// TIA Portal V18 export
// export: Created 2026-06-12T02:00:00Z, ExportSetting WithDefaults, DisplayName Totally Integrated Automation Portal, DisplayVersion V18, DisplayName TIA Portal Openness, DisplayVersion V18
TagTable "AI_B5_Tags"
  AI_B5_CA_Fan_Motor_DE_Temp : Real  (PLC tag AI_B5_CA_Fan_Motor_DE_Temp, HMI_Connection_1, 1 s)   // TEMP 50-80 °C
  AI_B5_CA_Fan_Motor_NDE_Temp : Real  (PLC tag AI_B5_CA_Fan_Motor_NDE_Temp, HMI_Connection_1, 1 s)   // TEMP 50-80 °C
  AI_B5_CA_Fan_DE_Temp : Real  (PLC tag AI_B5_CA_Fan_DE_Temp, HMI_Connection_1, 1 s)   // TEMP 50-80 °C
  AI_B5_CA_Fan_NDE_Temp : Real  (PLC tag AI_B5_CA_Fan_NDE_Temp, HMI_Connection_1, 1 s)   // TEMP 50-80 °C
  AI_B5_CA_Fan_DE_Vib : Real  (PLC tag AI_B5_CA_Fan_DE_Vib, HMI_Connection_1, 1 s)   // COUNT 0-10 mm/s
  AI_B5_CA_Fan_NDE_Vib : Real  (PLC tag AI_B5_CA_Fan_NDE_Vib, HMI_Connection_1, 1 s)   // COUNT 0-10 mm/s
  AI_B5_SP_700FN03 : Real  (PLC tag AI_B5_SP_700FN03, HMI_Connection_1, 1 s)   // FLOW 100-200 L/h
  AI_B5_SP_700HES01 : Real  (PLC tag AI_B5_SP_700HES01, HMI_Connection_1, 1 s)   // FLOW 100-200 L/h
  AI_B5_SP_700DA4 : Real  (PLC tag AI_B5_SP_700DA4, HMI_Connection_1, 1 s)   // FREQ 20-30 Hz
  AI_B5_SP_700DA6 : Real  (PLC tag AI_B5_SP_700DA6, HMI_Connection_1, 1 s)   // FREQ 20-30 Hz
  AI_B5_SP_700DA7 : Real  (PLC tag AI_B5_SP_700DA7, HMI_Connection_1, 1 s)   // FREQ 20-30 Hz
  AI_B5_SP_700FN2_DA1 : Real  (PLC tag AI_B5_SP_700FN2_DA1, HMI_Connection_1, 1 s)   // FREQ 20-30 Hz
  AI_B5_Sep_Motor_Top_Temp : Real  (PLC tag AI_B5_Sep_Motor_Top_Temp, HMI_Connection_1, 1 s)   // TEMP 50-80 °C
  AI_B5_Sep_Bottom_Bear_Temp : Real  (PLC tag AI_B5_Sep_Bottom_Bear_Temp, HMI_Connection_1, 1 s)   // TEMP 50-80 °C
  AI_B5_Trend_Val_1 : Real  (PLC tag AI_B5_Trend_Val_1, HMI_Connection_1, 1 s)   // PERCENT 0-100 %
  AI_B5_Trend_Val_2 : Real  (PLC tag AI_B5_Trend_Val_2, HMI_Connection_1, 1 s)   // PERCENT 0-100 %
  AI_B5_Trend_Val_3 : Real  (PLC tag AI_B5_Trend_Val_3, HMI_Connection_1, 1 s)   // PERCENT 0-100 %
  AI_B5_700FN03_RPM : Real  (PLC tag AI_B5_700FN03_RPM, HMI_Connection_1, 1 s)   // RPM 800-1200 RPM
  AI_B5_700HES01_Flow : Real  (PLC tag AI_B5_700HES01_Flow, HMI_Connection_1, 1 s)   // FLOW 100-200 L/h
  AI_B5_700FN10_Speed : Real  (PLC tag AI_B5_700FN10_Speed, HMI_Connection_1, 1 s)   // FREQ 20-30 Hz
  AI_B5_700CM01_Current : Real  (PLC tag AI_B5_700CM01_Current, HMI_Connection_1, 1 s)   // CURRENT 50-200 A
  AI_B5_Lub_Stop_Time : Real  (PLC tag AI_B5_Lub_Stop_Time, HMI_Connection_1, 1 s)   // COUNT 0-300 Sec
  AI_B5_Main_Drive_ReHealth : Real  (PLC tag AI_B5_Main_Drive_ReHealth, HMI_Connection_1, 1 s)   // COUNT 0-300 Sec
  AI_B5_CM_LRS_IN : Real  (PLC tag AI_B5_CM_LRS_IN, HMI_Connection_1, 1 s)   // TEMP 50-80 °C
  AI_B5_CM_LRS_OUT : Real  (PLC tag AI_B5_CM_LRS_OUT, HMI_Connection_1, 1 s)   // TEMP 50-80 °C
  AI_B5_CM_Mill_Oil_Temp : Real  (PLC tag AI_B5_CM_Mill_Oil_Temp, HMI_Connection_1, 1 s)   // TEMP 50-80 °C
  AI_B5_CM_OilTrun_BER_Temp : Real  (PLC tag AI_B5_CM_OilTrun_BER_Temp, HMI_Connection_1, 1 s)   // TEMP 50-80 °C
  AI_B5_CM_OilTrun_BER2_Temp : Real  (PLC tag AI_B5_CM_OilTrun_BER2_Temp, HMI_Connection_1, 1 s)   // TEMP 50-80 °C
  AI_B5_CM_OilPinion_BER_Temp : Real  (PLC tag AI_B5_CM_OilPinion_BER_Temp, HMI_Connection_1, 1 s)   // TEMP 50-80 °C
  AI_B5_CM_GB_IL_Shaft_BER : Real  (PLC tag AI_B5_CM_GB_IL_Shaft_BER, HMI_Connection_1, 1 s)   // TEMP 50-80 °C
  AI_B5_CM_Running_Hours : Real  (PLC tag AI_B5_CM_Running_Hours, HMI_Connection_1, 1 s)   // COUNT 0-8760 Hr
  AI_B5_CM_PS1_1_KG : Real  (PLC tag AI_B5_CM_PS1_1_KG, HMI_Connection_1, 1 s)   // PRESSURE 7-8 bar
  AI_B5_CM_PS1_2_KG : Real  (PLC tag AI_B5_CM_PS1_2_KG, HMI_Connection_1, 1 s)   // PRESSURE 7-8 bar
  AI_B5_NIBS_Value : Real  (PLC tag AI_B5_NIBS_Value, HMI_Connection_1, 1 s)   // CURRENT 50-200 A
  AI_B5_800DC1_Temp : Real  (PLC tag AI_B5_800DC1_Temp, HMI_Connection_1, 1 s)   // TEMP 50-80 °C
  AI_B5_800DC2_Temp : Real  (PLC tag AI_B5_800DC2_Temp, HMI_Connection_1, 1 s)   // TEMP 50-80 °C
  AI_B5_800FN1_Speed : Real  (PLC tag AI_B5_800FN1_Speed, HMI_Connection_1, 1 s)   // FREQ 20-30 Hz
  AI_B5_800FN2_Speed : Real  (PLC tag AI_B5_800FN2_Speed, HMI_Connection_1, 1 s)   // FREQ 20-30 Hz
  AI_B5_800YF1_Flow : Real  (PLC tag AI_B5_800YF1_Flow, HMI_Connection_1, 1 s)   // FLOW 100-200 L/h
  AI_B5_800YF2_Flow : Real  (PLC tag AI_B5_800YF2_Flow, HMI_Connection_1, 1 s)   // FLOW 100-200 L/h
  AI_B5_Silo1_Level_Bar1 : Real  (PLC tag AI_B5_Silo1_Level_Bar1, HMI_Connection_1, 1 s)   // LEVEL 0-100 %
  AI_B5_Silo1_Level_Bar2 : Real  (PLC tag AI_B5_Silo1_Level_Bar2, HMI_Connection_1, 1 s)   // LEVEL 0-100 %
  AI_B5_Silo2_Level_Bar1 : Real  (PLC tag AI_B5_Silo2_Level_Bar1, HMI_Connection_1, 1 s)   // LEVEL 0-100 %
  AI_B5_Silo2_Level_Bar2 : Real  (PLC tag AI_B5_Silo2_Level_Bar2, HMI_Connection_1, 1 s)   // LEVEL 0-100 %
  AI_B5_700FN01_Speed : Real  (PLC tag AI_B5_700FN01_Speed, HMI_Connection_1, 1 s)   // FREQ 20-30 Hz
  AI_B5_700FN02_Speed : Real  (PLC tag AI_B5_700FN02_Speed, HMI_Connection_1, 1 s)   // FREQ 20-30 Hz
  AI_B5_700AS07_Speed : Real  (PLC tag AI_B5_700AS07_Speed, HMI_Connection_1, 1 s)   // FREQ 20-30 Hz
  AI_B5_700AS08_Flow : Real  (PLC tag AI_B5_700AS08_Flow, HMI_Connection_1, 1 s)   // FLOW 100-200 L/h
  AI_B5_700FN09_Speed : Real  (PLC tag AI_B5_700FN09_Speed, HMI_Connection_1, 1 s)   // FREQ 20-30 Hz
  AI_B5_700SFM01_Speed : Real  (PLC tag AI_B5_700SFM01_Speed, HMI_Connection_1, 1 s)   // FREQ 20-30 Hz
  AI_B5_700DA1_Flow : Real  (PLC tag AI_B5_700DA1_Flow, HMI_Connection_1, 1 s)   // FLOW 100-200 L/h
  AI_B5_700DA4_Flow : Real  (PLC tag AI_B5_700DA4_Flow, HMI_Connection_1, 1 s)   // FLOW 100-200 L/h
  AI_B5_700DA6_Temp : Real  (PLC tag AI_B5_700DA6_Temp, HMI_Connection_1, 1 s)   // TEMP 50-80 °C
  AI_B5_700DA7_Temp : Real  (PLC tag AI_B5_700DA7_Temp, HMI_Connection_1, 1 s)   // TEMP 50-80 °C
  AI_B5_700BL1_Load : Real  (PLC tag AI_B5_700BL1_Load, HMI_Connection_1, 1 s)   // CURRENT 50-200 A
  AI_B5_700BL2_Load : Real  (PLC tag AI_B5_700BL2_Load, HMI_Connection_1, 1 s)   // CURRENT 50-200 A
  AI_B5_700AS9_Flow : Real  (PLC tag AI_B5_700AS9_Flow, HMI_Connection_1, 1 s)   // FLOW 100-200 L/h
  AI_B5_700FN13_Speed : Real  (PLC tag AI_B5_700FN13_Speed, HMI_Connection_1, 1 s)   // FREQ 20-30 Hz
